{attribute 'qualified_only'}
{attribute 'strict'}
{attribute 'to_string'}
TYPE TASK_TRANSITION_STATE :
(
	IDLE := 0,
	START,
	IN_PROGRES,	
	COMPETE
);
END_TYPE

(* stored: Version 1.1.0.1
   DUT TASK_TRANSITION_STATE: Id {8afe1cbb-da7f-4187-86ff-4bdc93959f0f} *)
